{attribute 'qualified_only'}
{attribute 'strict'}
TYPE StationList_e :
(
    ST105,
    ST110,
    ST115,
    ST120,
    ST125,
    ST130,
    ST135,
    ST140,
    ST145,
    ST150,
    ST155,
    ST160,
    ST165,
    ST170,
    //ST174 // is ignored because it is a waiting station
    ST175,
    ST176,
    ST180,
    ST185,
	_max
);
END_TYPE

(* stored: Version 1.1.0.1, ProductVersion 3.1.4024.6
   EnumerationTextList StationList_e: Id {7673be44-2b38-4ec9-b4a3-b2cf34b502a2} *)
